FUNCTION_BLOCK V_SENSE (* VSTYLE presence sensor *)
  (* Standard: 61499-1; Classification: Simulation *)
  (* Version 0.2, 2005-06-01, JHC, Holobloc Inc, Recompiled with new emitter. *)
  (* Version 0.1, 2002-04-20, JHC, Rockwell Automation, Moved to fb.rt.mva *)
  (* Version 0.0, 2002-04-10, JHC, Rockwell Automation *)
  (* Compiler header: package fb.rt.mva; *)
  (* Compiler Java IBM VisualAge 3.0 *)
  (* Compiler Java IBM Jikes 1.06 *)
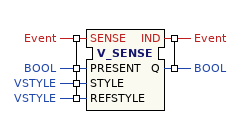
  EVENT_INPUT
    SENSE WITH PRESENT, STYLE, REFSTYLE; (* Input change notification *)
  END_EVENT
  EVENT_OUTPUT
    IND WITH Q; (* Output change indication *)
  END_EVENT
  VAR_INPUT
    PRESENT : BOOL; (* Workpiece is present *)
    STYLE : VSTYLE; (* Workpiece style *)
    REFSTYLE : VSTYLE; (* Style to be sensed *)
  END_VAR
  VAR_OUTPUT
    Q : BOOL; (* Workpiece is present and STYLE matches REFSTYLE *)
  END_VAR
  ALGORITHM SENSE IN Java:
boolean newq = PRESENT.value & (STYLE.equals(REFSTYLE));
if(newq != Q.value){
   Q.value = newq;
   IND.serviceEvent(this);}
  END_ALGORITHM
END_FUNCTION_BLOCK
